Staubli VAL3: getPoint.pgx

public program getPoint(point& x_pPoint[] (dimensions=1), bool x_bCycle (dimensions=1), num x_nIndex (dimensions=1))
  local string l_sItem
  local tool l_tTool
  local joint l_jJoint
begin
  // check the point
  link(x_pPoint,world)
  // use the flange
  l_tTool=flange
  // give back the point
  call getJointData(l_jJoint,l_tTool,x_bCycle,x_nIndex)
  x_pPoint=jointToPoint(l_tTool,world,l_jJoint)
end
